// TIA Portal V17 export
// export: Created 2024-08-09T12:53:13.6043815Z, ExportSetting WithDefaults, DisplayName Totally Integrated Automation Portal, DisplayVersion V17 Update 7, DisplayName TIA Portal Openness, DisplayVersion V17 Update 7, DisplayName TIA Portal Version Control Interface, DisplayVersion V17, DisplayName STEP 7 Professional, DisplayVersion V17 Update 7, DisplayName STEP 7 Safety, DisplayVersion V17 Update 6, DisplayName WinCC Professional, DisplayVersion V17 Update 7
VAR_GLOBAL   // PLC tag table "TREMIE_TRANS"
END_VAR
VAR_GLOBAL CONSTANT   // user constants
   NIV_TREMIE_TRANS_DEBUT_LOT : USInt := 1;
   NIV_TREMIE_TRANS_AUT_REMP : USInt := 10;
   NIV_TREMIE_TRANS_PRES_PRD : USInt := 20;
   NIV_TREMIE_TRANS_LANCE_EXTRACT : USInt := 25;
   NIV_TREMIE_TRANS_DEM_EXTRACT : USInt := 30;
   NIV_TREMIE_TRANS_PM : USInt := 40;
   NIV_TREMIE_TRANS_NB : USInt := 45;
   NIV_TREMIE_TRANS_VID_DEPUIS_X_SEC : USInt := 50;
   NIV_TREMIE_TRANS_NIVEAU_BAS : USInt := 60;
   NIV_TREMIE_TRANS_TEMPO_MINI : USInt := 70;
   NIV_TREMIE_TRANS_FIN_PM : USInt := 80;
   NIV_TREMIE_TRANS_DEBUT_VIDANGE : USInt := 90;
   NIV_TREMIE_TRANS_FIN_LOT : USInt := 255;
END_VAR
